TYPE TcoCr800_Inputs_v_1_x_x :
STRUCT
	Inputs AT %I* : ARRAY[0..63] OF BYTE;
END_STRUCT
END_TYPE

(* stored: Version 1.1.0.1, ProductVersion 3.1.4024.12
   DUT TcoCr800_Inputs_v_1_x_x: Id {b4d79663-a5a8-0b80-0bb0-4319f86ddfa4} *)
